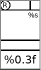
VISUALIZATION _VISU_WorkerDefGrid_small  // 41x70
VAR_IN_OUT
	m_Inst : FB_WorkerDefGrid;
END_VAR
    Rectangle (0,0 40x40), tooltip "%s"
        p4168582468: m_Inst._name
        OnMouseClick: change screen: AssignExpression m_Inst._sVisuName
    Rectangle (0,50 40x20), "%0.3f", tooltip "WorkerPosition", text variable: m_Inst.fPosition, colour toggle: m_Inst._fWorkerPosition = 0
        OnMouseClick: write the text variable via Default
    Rectangle (0,0 30x10), tooltip "Working pCT", colour toggle: m_Inst.bAttached
    Rectangle (1,10 40x10), "%s", text variable: m_Inst._name
    Rectangle (0,40 40x10), tooltip "Enable"
        toggle m_Inst.bEnable
    Ellipse (0,0 10x10), "R"
        tap m_Inst._bForceRelease
    Rectangle (30,0 10x10), tooltip "error: %d", colour toggle: m_Inst.bError
        p4168582468: m_Inst.nError
END_VISUALIZATION

(* stored: Version 1.1.0.1, ProductVersion 3.1.4024.3
   Visu _VISU_WorkerDefGrid_small: Id {e4f5b659-9e66-4187-a0fe-9dea7a61c02d} *)
